// SIMATIC S7-200 project (STEP 7-Micro/WIN), CPU 224XP REL 02.01

SYMBOL_TABLE USER1
star             I0.0
s_top            I0.1
bom1             Q0.0
bom2             Q0.1
bien             M0.0
muc_be_tren      I0.2
END_SYMBOL_TABLE

ORGANIZATION_BLOCK MAIN:OB1
TITLE=PROGRAM COMMENTS
BEGIN
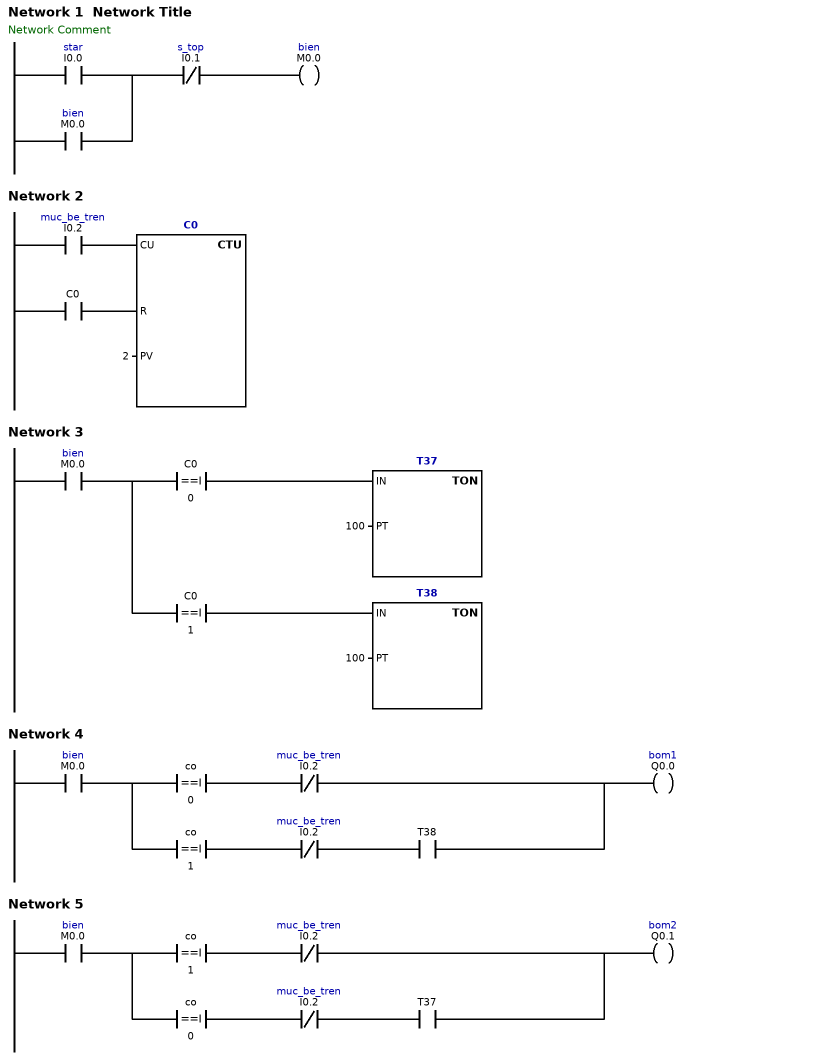
Network 1 // Network Title
// Network Comment
LD     star:I0.0
O      bien:M0.0
AN     s_top:I0.1
=      bien:M0.0
Network 2
LD     muc_be_tren:I0.2
LD     C0
CTU    C0, 2
Network 3
LD     bien:M0.0
LPS
AW=    C0, 0
TON    T37, 100
LPP
AW=    C0, 1
TON    T38, 100
Network 4
// (network saved uncompiled; LAD cells follow)
// row 0: c0 -| |- bien:M0.0 v  c1 -|==I|- co, 0  c2 -|/|- muc_be_tren:I0.2  c3 --  c4 -- v  c5 -( ) bom1:Q0.0
// row 1: c0 ^  c1 -|==I|- co, 1  c2 -|/|- muc_be_tren:I0.2  c3 -| |- T38  c4 -- ^
Network 5
// (network saved uncompiled; LAD cells follow)
// row 0: c0 -| |- bien:M0.0 v  c1 -|==I|- co, 1  c2 -|/|- muc_be_tren:I0.2  c3 --  c4 -- v  c5 -( ) bom2:Q0.1
// row 1: c0 ^  c1 -|==I|- co, 0  c2 -|/|- muc_be_tren:I0.2  c3 -| |- T37  c4 -- ^
END_ORGANIZATION_BLOCK
